   //adapt the calculated random number to the given number span
   #tempNormReal := NORM_X(MIN := #MIN_UDINT, VALUE := #tempRandomValue, MAX := #MAX_UDINT);
   // #LGF_RandomReal := SCALE_X(MIN := #minValue, VALUE := #tempNormReal, MAX := #maxValue);
   #LGF_RandomReal := #tempNormReal * (#maxValue - #minValue) + #minValue;

   #status := #NO_ERROR;
END_FUNCTION

FUNCTION "LRamp_001" : Void   // FC20401, SCL
TITLE = LRamp_001
{ S7_Optimized_Access := 'TRUE' }
AUTHOR : CISDI
FAMILY : TECHNO
VERSION : 0.1
// 1. linear ramp output to setvalue with a fixed acceleration
// 2. slope of ramp output = i_R_Acc
// 3. i_R_Tcyc and i_R_Acc must be >0.0
   VAR_INPUT
      i_R_Tcyc : Real;   // OB cycle time (ms)
      i_R_SetValue : Real;   // ramp input setvalue [unit]
      i_R_Acc : Real;   // acceleration set [unit/s]
   END_VAR
   VAR_OUTPUT
      o_B_ParamErr : Bool;   // parameter error
      o_B_EndRmp : Bool;   // ramp output reached setvalue
      o_B_ZeroRmp : Bool;   // ramp output =0
      o_B_Acc : Bool;   // ramp output is increasing
      o_B_Dec : Bool;   // ramp output is decreasing
      o_R_Acc : Real;   // accelerate ( [unit of setvalue]/s)
   END_VAR
   VAR_IN_OUT
      io_R_OutRmp : Real;   // ramp output [unit]
   END_VAR
   VAR_TEMP
      tmp_R_Step : Real;   // ramp step
      tmp_R_Delta : Real;   // delta = setvalue - rampoutput
      tmp_R_DeltaAbs : Real;   // abs(delta)
      tmp_R_OutRmp_Pre : Real;   // ramp output of previous scan
   END_VAR
BEGIN
   (*
   // ===========================================================================
   // CISDI
   // (c)Copyright (2017) All Rights Reserved
   // ---------------------------------------------------------------------------
   // Library: (LPM)
   // Tested with: (S7-1500)
   // Engineering: TIA Portal (V13)
   // Restrictions:
   // 1.must be called in cyclic interrupt OB (eg.OB30)
   // Requirements: ( )
   // Functionality: 
   // 1. linear ramp output to setvalue with a fixed acceleration
   // 2. slope of ramp output = i_R_Acc
   // 3. i_R_Tcyc and i_R_Acc must be >0.0
   // ---------------------------------------------------------------------------
   // Change log table:
   // Version     Date          Expert in charge    Changes applied
   // 00.00.01    27.03.2017    002897              First released version
   // ===========================================================================
   *)
   // parameter check
   IF #i_R_Tcyc <= 0.0 OR #i_R_Acc <= 0.0 THEN
       // parameter is error
       #o_B_ParamErr := 1;
       #io_R_OutRmp := 0.0;
       #o_R_Acc := 0.0;
       #o_B_EndRmp := 0;
       #o_B_ZeroRmp := 0;
       #o_B_Acc := 0;
       #o_B_Dec := 0;
       RETURN;
   ELSE
       // set ramp output to setvalue
       #tmp_R_OutRmp_Pre := #io_R_OutRmp;
       #tmp_R_Delta := #i_R_SetValue - #io_R_OutRmp;
       #tmp_R_DeltaAbs := ABS(IN := #tmp_R_Delta);
       #tmp_R_Step := #i_R_Acc * #i_R_Tcyc * 0.001;
       IF #tmp_R_DeltaAbs < #tmp_R_Step THEN
           #io_R_OutRmp := #i_R_SetValue;
       ELSIF #tmp_R_Delta >= #tmp_R_Step THEN
           #io_R_OutRmp := #io_R_OutRmp + #tmp_R_Step;
       ELSE
           #io_R_OutRmp := #io_R_OutRmp - #tmp_R_Step;
       END_IF;

       // acceleration
       #o_R_Acc := (#io_R_OutRmp - #tmp_R_OutRmp_Pre) / (#i_R_Tcyc * 0.001);

       // status of ramp
       #o_B_EndRmp := #io_R_OutRmp = #i_R_SetValue;
       #o_B_ZeroRmp := #io_R_OutRmp = 0.0;
       #o_B_Acc := #io_R_OutRmp > #tmp_R_OutRmp_Pre;
       #o_B_Dec := #io_R_OutRmp < #tmp_R_OutRmp_Pre;

   END_IF;
END_FUNCTION

FUNCTION "DeadBand_Real" : Void   // FC30005, SCL
{ S7_Optimized_Access := 'TRUE' }
VERSION : 0.1
   VAR_INPUT
      i_R_X : Real;
      i_R_DBWidth : Real;
   END_VAR
   VAR_OUTPUT
      o_R_Y : Real;
   END_VAR
   VAR_TEMP
      i_R_AbsX : Real;
      i_R_AbsDBWidth : Real;
   END_VAR
BEGIN
   #i_R_AbsX := ABS(#i_R_X);
   #i_R_AbsDBWidth := ABS(#i_R_DBWidth);
   IF #i_R_AbsX > #i_R_AbsDBWidth AND #i_R_X >= 0 THEN
       #o_R_Y := #i_R_X - #i_R_AbsDBWidth;
   ELSIF #i_R_AbsX > #i_R_AbsDBWidth AND #i_R_X < 0 THEN
       #o_R_Y := #i_R_X + #i_R_AbsDBWidth;
   ELSE
       #o_R_Y := REAL#0.0;
   END_IF;
END_FUNCTION

// ===== library types =====

// folder: 4 Math operations

FUNCTION "LGF_RandomBasic" : Real   // FC10038, SCL
{ S7_Optimized_Access := 'TRUE' }
   VAR_TEMP
      tempTime : DTL;   // System time
      tempTimeStatus : Int;   // Status of the instruction RD_SYS_T
      tempRandomValue : UDInt;   // Random-start-value
   END_VAR
   // Ret_Val : Ret_Val
   VAR CONSTANT
      MIN_UDINT : UDInt := 0;   // UDInt lower value range
      MAX_UDINT : UDInt := 4294967295;   // UDInt upper value range
   END_VAR
BEGIN
   //=============================================================================
   // Siemens AG
   // (c)Copyright 2017
   //-----------------------------------------------------------------------------
   // Library:       LGF (Library General Functions)
   // Tested with:   CPU1212C DC/DC/DC FW:V4.2
   // Engineering:   TIA Portal V14 Upd 1
   // Restrictions:  -
   // Requirements:  PLC (S7-1200 / S7-1500)
   // Functionality: This function generates random numbers. 0.0 <= REAL <= 1.0
   //                (Datatype Real)
   //-----------------------------------------------------------------------------
   // Change log table:
   // Version  Date        In charge/Changes applied
   // 01.00.00 27.01.2017  Siemens Industry Online Support
   //                      First released version
   //-----------------------------------------------------------------------------
   //Status Codes: -
   //=============================================================================

   //Read system time
   #tempTimeStatus := RD_SYS_T(#tempTime);

   //Callculate a random-start-value depending on the time
   #tempRandomValue.%B3 := #tempTime.NANOSECOND.%B0;
   #tempRandomValue.%B2 := #tempTime.NANOSECOND.%B1;
   #tempRandomValue.%B1 := #tempTime.NANOSECOND.%B2;
   #tempRandomValue.%B0 := #tempTime.NANOSECOND.%B3;

   //Norm the calculated random number: 0.0 <= #LGF_RandomBasic <= 1.0
   #LGF_RandomBasic := NORM_X(MIN := #MIN_UDINT, VALUE := #tempRandomValue, MAX := #MAX_UDINT);
END_FUNCTION

// folder: 5 Data handling

FUNCTION_BLOCK "LGF_FIFO"   // FB10017, SCL
{ S7_Optimized_Access := 'TRUE' }
   VAR_INPUT
      execute : Bool;   // The instruction is executed when a positive signal edge is detected at the "request" parameter.
      mode : Bool;   // 0 = The first entry in the ring buffer is returned. 1 = An entry is written at the last position in the ring buffer.
      initialValue : Variant;   // Value with which the ARRAY of the ring buffer is initialized.
      resetBuffer : Bool;
   END_VAR
   VAR_OUTPUT
      done : Bool;
      error : Bool;
      statusID : UInt;
      status : Word;   // Status information
   END_VAR
   VAR_IN_OUT
      item : Variant;   // The entry that is either returned from the ring buffer or written to the ring buffer
      buffer : Variant;   // An ARRAY that is used as a ring buffer.
   END_VAR
   VAR
      statEdgeupm : Bool;   // Edge memory bit in which the RLO of the previous query is saved.
      statFirstItemIndex : Int := -1;   // Index of the oldest entry in the ring buffer
      statNextEmptyItemIndex : Int := 0;   // Index of the next free entry in the ring buffer
   END_VAR
   VAR_TEMP
      tempEdgeup : Bool;   // Result of edge evaluation
      tempInternalError : Int;   // Error information
      tempNewFirstItemIndex : Int;   // Variable index
      tempNewNextEmptyItemIndex : Int;   // Variable index
      tempPufferSize : UDInt;   // Number of ARRAY elements in the ring buffer
      tempSizeCounter : Int;
   END_VAR
   VAR CONSTANT
      NO_ERROR : Word := 16#0000;
      NO_CURRENT_JOBS : Word := 16#7000;
      BUFFER_EMPTY : Word := 16#8001;
      BUFFER_FULL : Word := 16#8002;
      NO_ARRAY : Word := 16#8200;
      WRONG_TYPE_1 : Word := 16#8201;
      WRONG_TYPE_2 : Word := 16#8202;
      INDEX_IN_ARRAY_LIMITS_1 : Word;
      INDEX_IN_ARRAY_LIMITS_2 : Word;
      ERROR_IN_THIS_BLOCK : UInt := 1;
      ERROR_MOVE_BLK_VARIANT : UInt := 2;
      NEXT_TASK_TO_EXECUTE : Bool := false;
      BUFFER_IS_EMPTY : Int := -1;
      BUFFER_CONTAINS_ARRAY : Int := 0;
      NO_INTERNAL_ERROR : Int := 0;
      BUFFER_INITIALIZED : Int := -1;
      RESET : Bool := true;
   END_VAR
BEGIN
   //=============================================================================
   // SIEMENS AG
   // (c)Copyright 2017
   //-----------------------------------------------------------------------------
   // Library:       LGF (Library General Functions)
   // Tested with:   CPU1212C DC/DC/DC FW:V4.2
   // Engineering:   TIA Portal V14
   // Restrictions:  -
   // Requirements:  PLC (S7-1200 / S7-1500)
   // Functionality: FIFO(First In First Out)-functionblock
   //-----------------------------------------------------------------------------
   // Change log table:
   // Version  Date        Expert in charge / Changes applied
   // 01.00.00 19.08.2015  Siemens Industry Online Support
   //                      First released version
   // 01.00.01 16.11.2015  Siemens Industry Online Support
   //                      Bug fix resetBuffer
   // 01.00.02 02.01.2017  Siemens Industry Online Support
   //                      Upgrade: TIA Portal V14 Update 1
   //=============================================================================

   //This program code section is only executed once after a negative signal edge.
   IF #execute = false AND #statEdgeupm = true THEN
     #done := false;
     // If no error occurred during program execution, the error code "0000" is output.  
     #error := false;
     #statusID := #ERROR_IN_THIS_BLOCK;
     #status := #NO_CURRENT_JOBS;
   END_IF;

   //This program code section is only executed once after a positive signal edge.
   //IF there is no change in the signal state OF the result OF logic operation,
   //the program processing OF the "FIFOQueue" FB is terminated.

   IF #execute <> true OR #statEdgeupm <> false THEN
     #statEdgeupm := #execute;
     RETURN;
   END_IF;
   #statEdgeupm := #execute;

   // ------Validation of whether all parameter inputs are valid.----

   //This program code section checks whether the ring #buffer is an ARRAY.
   //IF so, the number OF the ARRAY elements is read out.
   //IF it is NOT an ARRAY, the program execution is terminated at this point
   //AND the status code "8200" is output.

   IF NOT (IS_ARRAY(#buffer)) THEN
     #error := true;
     #statusID := #ERROR_IN_THIS_BLOCK;
     #status := #NO_ARRAY;
     RETURN;
   ELSE
     #tempPufferSize := CountOfElements(#buffer);
   END_IF;

   //This program code section checks whether the data type OF the ARRAY elements matches
   //the data type OF the entry (tag #item). IF the data types DO NOT match,
   //the program execution is terminated at this point AND the error code "8201" is output.

   IF NOT (TypeOf(#item) = TypeOfElements(#buffer)) THEN
     #error := true;
     #statusID := #ERROR_IN_THIS_BLOCK;
     #status := #WRONG_TYPE_1;
     RETURN;
   END_IF;

   //This program code section checks whether the initial value OF the ring #buffer
   //matches the entry (tag #item). IF the data types DO NOT match,
   //the program execution is terminated at this point
   //AND the error code "8202" is output. *)

   IF NOT (TypeOf(#item) = TypeOf(#initialValue)) THEN
     #error := true;
     #statusID := #ERROR_IN_THIS_BLOCK;
     #status := #WRONG_TYPE_2;
     RETURN;
   END_IF;

   //This program code section checks whether the variable indices are within the ARRAY limits.
   //IF they are NOT, the program execution is terminated at this point
   //AND either error code "8601" OR "8602" is output depending on the index. *)

   IF (#statNextEmptyItemIndex >= #tempPufferSize) THEN
     #error := true;
     #statusID := #ERROR_IN_THIS_BLOCK;
     #status := #INDEX_IN_ARRAY_LIMITS_1;
     RETURN;
   END_IF;

   IF (#statFirstItemIndex >= #tempPufferSize) THEN
     #error := true;
     #statusID := #ERROR_IN_THIS_BLOCK;
     #status := #INDEX_IN_ARRAY_LIMITS_2;
     RETURN;
   END_IF;


   //If reset is "TRUE" the buffer and their  counters are resetted
   IF #resetBuffer = #RESET THEN
     #statFirstItemIndex := -1;
     #statNextEmptyItemIndex := 0;

     FOR #tempSizeCounter := 0 TO UDINT_TO_INT(#tempPufferSize - 1) DO

       #tempInternalError := MOVE_BLK_VARIANT(SRC := #initialValue,
                                              COUNT := 1,
                                              SRC_INDEX := 0,
                                              DEST_INDEX := #tempSizeCounter,
                                              DEST => #buffer);
     END_FOR;
     IF (#tempInternalError <> #NO_INTERNAL_ERROR) THEN
       #error := true;
       #statusID := #ERROR_MOVE_BLK_VARIANT;
       #status := INT_TO_WORD(#tempInternalError);
     END_IF;
     RETURN;
   END_IF;

   //-----------Program code execution, depending on the Mode parameter-------------
   // The execution of the instructions depends on the signal state of the Mode parameter.

   IF #mode = #NEXT_TASK_TO_EXECUTE THEN


     // If the Mode parameter has the signal state "0",
     // the first entry from the passed ring buffer is returned.

     //this program code section checks whether the ring #buffer is empty.
     //IF this is the CASE, program execution is terminated at this point
     //AND the error code "8001" is output. *)

     IF (#statFirstItemIndex = #BUFFER_IS_EMPTY) THEN
       #error := true;
       #statusID := #ERROR_IN_THIS_BLOCK;
       #status := #BUFFER_EMPTY;
       RETURN;
     END_IF;


     // This program code section returns the first entry of the ring buffer.

     #tempInternalError := MOVE_BLK_VARIANT(SRC := #buffer,
                                            COUNT := 1,
                                            SRC_INDEX := #statFirstItemIndex,
                                            DEST_INDEX := 0,
                                            DEST => #item);

     IF (#tempInternalError = #BUFFER_CONTAINS_ARRAY) THEN

       //This program code section checks whether the ring #buffer contains ARRAY elements.
       //IF it does, the first entry is passed further on
       //AND the index is incremented BY 1. *)

       #tempInternalError := MOVE_BLK_VARIANT(SRC := #initialValue,
                                              COUNT := 1,
                                              SRC_INDEX := 0,
                                              DEST_INDEX := #statFirstItemIndex,
                                              DEST => #buffer);

       // This program code section calculates the new index of the first entry.

       #tempNewFirstItemIndex := #statFirstItemIndex + 1;
       #tempNewFirstItemIndex := #tempNewFirstItemIndex MOD UDINT_TO_INT(#tempPufferSize);

       // This program section checks whether the ring buffer is empty.        
       IF (#statNextEmptyItemIndex = #tempNewFirstItemIndex) THEN
         // If the ring buffer is empty, the index is set to 0.            
         #statFirstItemIndex := -1;
         #statNextEmptyItemIndex := 0;
       ELSE
         // The index of the first entry is changed.            
         #statFirstItemIndex := #tempNewFirstItemIndex;
       END_IF;
     END_IF;
   ELSE

     // If the Mode parameter has the signal state "1", the entry is written to the passed ring buffer.

     //this program code section checks whether the ring #buffer is full.
     //IF this is the CASE, program execution is terminated at this point
     //AND the error code "8002" is output. *)

     IF (#statNextEmptyItemIndex = #statFirstItemIndex) THEN
       #error := true;
       #statusID := #ERROR_IN_THIS_BLOCK;
       #status := #BUFFER_FULL;
       RETURN;
     END_IF;

     // This program code section writes the entry to the ring buffer.   
     #tempInternalError := MOVE_BLK_VARIANT(SRC := #item,
                                            COUNT := 1,
                                            SRC_INDEX := 0,
                                            DEST_INDEX := #statNextEmptyItemIndex,
                                            DEST => #buffer);

     IF (#tempInternalError = #NO_INTERNAL_ERROR) THEN

       // This program code section increments the index by 1 and calculates the new empty entry index.        
       #tempNewNextEmptyItemIndex := #statNextEmptyItemIndex + 1;
       #tempNewNextEmptyItemIndex := #tempNewNextEmptyItemIndex MOD UDINT_TO_INT(#tempPufferSize);
       #statNextEmptyItemIndex := #tempNewNextEmptyItemIndex;

       //This program code section checks which index the "#firstItemIndex" tag has.
       //IF the number = -1, the ring buffer is initialized
       //AND the entry is written TO the ring #buffer.
       //Therefore, "0" must be assigned TO the tag.

       IF (#statFirstItemIndex = #BUFFER_INITIALIZED) THEN
         #statFirstItemIndex := 0;
       END_IF;
     END_IF;
   END_IF;

   //-------------------------Local error handling----------------------------
   //This program code section checks whether a "Local" #error has occurred.
   //IF This is the CASE, program execution is terminated at This point
   //AND the error code of MOV_BLK_VARIANT is output. *)

   IF (#tempInternalError <> #NO_INTERNAL_ERROR) THEN
     #error := true;
     #statusID := #ERROR_MOVE_BLK_VARIANT;
     #status := INT_TO_WORD(#tempInternalError);
     RETURN;
   END_IF;

   #done := true;
   #status := #NO_ERROR;
END_FUNCTION_BLOCK

FUNCTION_BLOCK "LGF_RingBuffer"   // FB10022, SCL
{ S7_Optimized_Access := 'TRUE' }
VERSION : 0.1
   VAR_INPUT
      write : Bool;   // With a rising edge newValue is written in ring buffer
      resetBuffer : Bool;   // Reset buffer
      newValue : Word;   // New Value
   END_VAR
   VAR_IN_OUT
      buffer : Array[*] of Word;   // Buffer
   END_VAR
   VAR
      statInitialized : Bool;   // -
      statElementReset : DInt;   // -
      statLowerLimit : DInt;   // -
      statUpperLimit : DInt;   // -
      statNumElements : UDInt;   // -
      statEdgeWrite : Bool;
   END_VAR
   VAR_TEMP
      tempRetVal : Int;   // -
   END_VAR
BEGIN
   //=============================================================================
   // Siemens AG
   // (c)Copyright 2017
   //-----------------------------------------------------------------------------
   // Library:       LGF (Library General Functions)
   // Tested with:   CPU1212C DC/DC/DC FW:V4.2
   // Engineering:   TIA Portal V14 SP1 Upd 5
   // Restrictions:  -
   // Requirements:  PLC (S7-1200 / S7-1500)
   // Functionality: Ring buffer-functionblock
   //-----------------------------------------------------------------------------
   // Change log table:
   // Version  Date        In charge / Changes applied
   // 01.00.00 03.07.2018  Siemens Industry Online Support
   //                      First released version
   //=============================================================================

   // Initialization
   IF (NOT #statInitialized)
   THEN
     #statLowerLimit := LOWER_BOUND(ARR := #buffer, DIM := 1);
     #statUpperLimit := UPPER_BOUND(ARR := #buffer, DIM := 1);
     #statNumElements := DINT_TO_UDINT(#statUpperLimit - #statLowerLimit + 1);
     #statInitialized := true;
   END_IF;

   IF (#write = TRUE)
     AND (NOT #statEdgeWrite)
     AND (NOT #resetBuffer)
   THEN
     // Move all elements but the last one one element up
     #tempRetVal := MOVE_BLK_VARIANT(SRC := #buffer,
                                     COUNT := #statNumElements - 1,
                                     SRC_INDEX := 0,
                                     DEST_INDEX := 1,
                                     DEST => #buffer);
     // Store new value to first element
     #buffer[#statLowerLimit] := #newValue;
   END_IF;

   IF (#resetBuffer = TRUE)
   THEN
     // Reset buffer
     FOR #statElementReset := #statLowerLimit TO #statUpperLimit DO
       // Statement section FOR
       #buffer[#statElementReset] := 0;
     END_FOR;

   END_IF;

   // Edge detection
   #statEdgeWrite := #write;
END_FUNCTION_BLOCK